Universal Robots PolyScope program: pulley_v2.urp

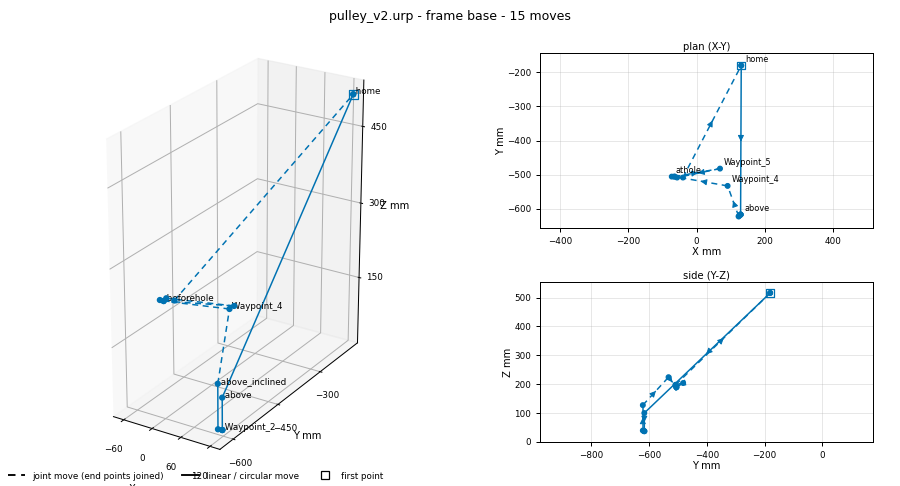
[picture p0: tool path of pulley_v2.urp in frame base, 15 of 23 moves have a stored position in this frame; points joined in program order, loops and branches not executed]
Program pulley_v2 (installation=default directory=/programs/wrs2020 createdIn=5.7.0.90932 lastSavedIn=5.7.0.90932 robotSerialNumber=20205500607)
Calibrated DH parameters: a=[0.000096, -0.337, -0.383372, 0.000118, 0.000015, 0]; d=[0.162724, 79.377998, -95.545185, 16.300583, 0.099689, 0.099499]; alpha=[1.569249, 0.003272, 0.005201, 1.570041, -1.570219, 0]; deltaTheta=[0, 0.65664, 5.410619, 0.215927, -0.000001, 0]
Robot Program (runOnlyOnce=true)
  MoveJ speed 180 deg/s, acceleration 80 deg/s^2 (useActiveTCP=true) feature=Base
    Waypoint home: TCP in base x=130.635 y=-180.692 z=515.97 mm, rx=-0.0117 ry=-3.1402 rz=-0.0315 rad; joints [89.951, -120.324, 80.212, -48.705, -89.957, -0.002] deg; TCP offset x=0 y=0 z=165 mm, rx=0 ry=0 rz=0 rad
  URCap Gripper (Robotiq_Grippers, Robotiq Inc.) dataModel(position=15.686274509803921, force=100.0, speed=100.0, positionInDouble=15.686274509803921, forceInDouble=100.0, speedInDouble=100.0, slaveIds=[9], blocking=true)
  MoveL speed 250 mm/s, acceleration 1200 mm/s^2 (useActiveTCP=true) feature=Base
    Waypoint above: TCP in base x=128.76 y=-616.729 z=99.924 mm, rx=1.2479 ry=2.8551 rz=-0.0099 rad; joints [89.154, -66.805, 95.766, -119.835, -88.426, 46.424] deg
    Waypoint Waypoint_2: TCP in base x=128.767 y=-616.702 z=37 mm, rx=1.2363 ry=2.8602 rz=-0.01 rad; joints [89.14, -62.119, 99.446, -128.198, -88.435, 45.999] deg; TCP offset x=0 y=0 z=165 mm, rx=0 ry=0 rz=0 rad
  URCap Gripper (Robotiq_Grippers, Robotiq Inc.) dataModel(position=100.0, force=0.0, speed=0.0, positionInDouble=100.0, forceInDouble=0.0, speedInDouble=0.0, slaveIds=[9], blocking=true)
  URCap Gripper (Robotiq_Grippers, Robotiq Inc.) dataModel(position=21.176470588235293, force=0.0, speed=0.0, positionInDouble=21.176470588235293, forceInDouble=0.0, speedInDouble=0.0, slaveIds=[9], blocking=true)
  MoveL speed 600 mm/s, acceleration 1200 mm/s^2 (useActiveTCP=true) feature=Base
    Waypoint Waypoint_3: TCP in base x=128.76 y=-616.729 z=37 mm, rx=-1.1525 ry=2.9078 rz=-0.0355 rad; joints [89.139, -62.118, 99.445, -128.202, -88.435, -43.999] deg; TCP offset x=0 y=0 z=165 mm, rx=0 ry=0 rz=0 rad
  URCap Gripper (Robotiq_Grippers, Robotiq Inc.) dataModel(position=100.0, force=0.0, speed=0.0, positionInDouble=100.0, forceInDouble=0.0, speedInDouble=0.0, slaveIds=[9], blocking=true)
  URCap Gripper (Robotiq_Grippers, Robotiq Inc.) dataModel(position=36.07843137254902, force=0.0, speed=0.0, positionInDouble=36.07843137254902, forceInDouble=0.0, speedInDouble=0.0, slaveIds=[9], blocking=true)
  MoveL speed 600 mm/s, acceleration 1200 mm/s^2 (useActiveTCP=true) feature=Base
    Waypoint Waypoint_2: TCP in base x=128.767 y=-616.702 z=37 mm, rx=1.2363 ry=2.8602 rz=-0.01 rad; joints [89.14, -62.119, 99.446, -128.198, -88.435, 45.999] deg; TCP offset x=0 y=0 z=165 mm, rx=0 ry=0 rz=0 rad
    Waypoint Waypoint_1: TCP in base x=123.202 y=-621.873 z=39.247 mm, rx=-1.1443 ry=-2.5469 rz=0.8367 rad; joints [100.881, -59.401, 111.69, -163.652, -118.977, 53.915] deg; TCP offset x=0 y=0 z=165 mm, rx=0 ry=0 rz=0 rad
  URCap Gripper (Robotiq_Grippers, Robotiq Inc.) dataModel(position=100.0, force=100.0, speed=100.0, positionInDouble=100.0, forceInDouble=100.0, speedInDouble=100.0, slaveIds=[9], blocking=true)
  MoveL speed 250 mm/s, acceleration 1200 mm/s^2 (useActiveTCP=true) feature=Base
    Waypoint above_inclined: TCP in base x=123.202 y=-621.873 z=127.29 mm, rx=-1.1443 ry=-2.5469 rz=0.8367 rad; joints [100.905, -68.525, 108.499, -151.362, -118.935, 53.865] deg
  SuppressedNode
    MoveJ speed 60 deg/s, acceleration 80 deg/s^2 (useActiveTCP=true) feature=Base
      Waypoint intermediate: motionParameters(blendRadius=0.05); TCP in base x=115.537 y=-464.392 z=278.491 mm, rx=2.1151 ry=-1.8246 rz=-0.1767 rad; joints [98.791, -95.537, 106.25, -108.287, -109.219, -91.027] deg
      Waypoint before_hole: TCP in base x=-57.686 y=-570.408 z=232.23 mm, rx=1.3727 ry=-1.1616 rz=-1.3181 rad; joints [97.319, -59.573, 88.654, -50.464, -171.504, -31.295] deg
  SuppressedNode
    MoveJ speed 60 deg/s, acceleration 80 deg/s^2 (useActiveTCP=true) feature=Base
      Waypoint at_hole: TCP in base x=-85.495 y=-570.408 z=232.23 mm, rx=1.3727 ry=-1.1616 rz=-1.3181 rad; joints [94.632, -61.815, 93.453, -62.169, -173.913, -40.501] deg; TCP offset x=0 y=0 z=165 mm, rx=0 ry=0 rz=0 rad
  SuppressedNode
    Force Frame feature=Joint_6_name; selection=[0, 0, 1, 0, 0, 0]; wrench=[0, 0, 10, 0, 0, 0]; limitsForce=[0.15, 0.15, 0.01, 1.047198, 1.047198, 1.047198]; limitsMotion=[0.1, 0.1, 0.1, 0.349066, 0.349066, 0.349066]
      MoveJ speed 60 deg/s, acceleration 80 deg/s^2 (useActiveTCP=true) feature=Base
        Waypoint turn_right (Relative): relativeFromPosition TCP in base x=-85.515 y=-570.41 z=232.207 mm, rx=1.3727 ry=-1.1616 rz=-1.3181 rad; joints [94.63, -61.813, 93.454, -62.171, -173.913, -40.501] deg; TCP offset x=0 y=0 z=165 mm, rx=0 ry=0 rz=0 rad; TCP in base x=-85.507 y=-570.407 z=232.241 mm, rx=0.846 ry=-1.441 rz=-0.7763 rad; joints [94.699, -63.491, 97.916, -73.842, -175.626, -8.792] deg
        Waypoint turn_left (Relative): relativeFromPosition TCP in base x=-85.52 y=-570.402 z=232.224 mm, rx=0.846 ry=-1.4411 rz=-0.7763 rad; joints [94.698, -63.49, 97.916, -73.843, -175.624, -8.792] deg; TCP in base x=-85.509 y=-570.398 z=232.173 mm, rx=1.3728 ry=-1.1615 rz=-1.3182 rad; joints [94.631, -61.811, 93.456, -62.169, -173.913, -40.501] deg
        Waypoint turn_left (Relative): relativeFromPosition TCP in base x=-85.52 y=-570.402 z=232.224 mm, rx=0.846 ry=-1.4411 rz=-0.7763 rad; joints [94.698, -63.49, 97.916, -73.843, -175.624, -8.792] deg; TCP in base x=-85.509 y=-570.398 z=232.173 mm, rx=1.3728 ry=-1.1615 rz=-1.3182 rad; joints [94.631, -61.811, 93.456, -62.169, -173.913, -40.501] deg
        Waypoint turn_right (Relative): relativeFromPosition TCP in base x=-85.515 y=-570.41 z=232.207 mm, rx=1.3727 ry=-1.1616 rz=-1.3181 rad; joints [94.63, -61.813, 93.454, -62.171, -173.913, -40.501] deg; TCP in base x=-85.507 y=-570.407 z=232.241 mm, rx=0.846 ry=-1.441 rz=-0.7763 rad; joints [94.699, -63.491, 97.916, -73.842, -175.626, -8.792] deg
  MoveJ speed 120 deg/s, acceleration 150 deg/s^2 (useActiveTCP=true) feature=Base
    Waypoint Waypoint_4: motionParameters(blendRadius=0.05); TCP in base x=90.784 y=-532.798 z=224.095 mm, rx=1.3194 ry=-2.4664 rz=0.0869 rad; joints [93.539, -87.4, 107.422, -121.697, -105.954, -54.416] deg
    Waypoint beforehole: TCP in base x=-64.521 y=-505.594 z=189.248 mm, rx=1.6358 ry=-1.672 rz=-0.8845 rad; joints [92.147, -76.667, 111.26, -118.048, -144.223, -83.204] deg
  MoveL speed 20 mm/s, acceleration 1200 mm/s^2 (useActiveTCP=true) feature=Base
    Waypoint athole: TCP in base x=-72.578 y=-505.587 z=189.228 mm, rx=1.6358 ry=-1.672 rz=-0.8845 rad; joints [91.256, -76.788, 111.802, -119.703, -144.314, -84.72] deg
  MoveL speed 250 mm/s, acceleration 1200 mm/s^2 (useActiveTCP=true) feature=Base
    MoveDirectionNode (selectedDirection=XMinus) feature=Base
      Until TOOL_CONTACT_DETECTION (allowActions=false retraction=0 decelerationAcceleration=3 decelerationAngularAcceleration=34.906585)
  Force Frame feature=Base; selection=[1, 1, 1, 0, 0, 0]; wrench=[-10, 0, 0, 0, 0, 0]; limitsForce=[0.01, 0.01, 0.01, 1.047198, 1.047198, 1.047198]; limitsMotion=[0.1, 0.1, 0.1, 0.349066, 0.349066, 0.349066]
    MoveL speed 50 mm/s, acceleration 200 mm/s^2 (useActiveTCP=true) feature=Base
      Waypoint rightturn (Relative): relativeFromPosition TCP in base x=-72.572 y=-505.592 z=189.212 mm, rx=1.6359 ry=-1.672 rz=-0.8845 rad; joints [91.257, -76.786, 111.802, -119.705, -144.314, -84.72] deg; TCP in base x=-72.593 y=-509.312 z=189.314 mm, rx=1.2962 ry=-1.7188 rz=-0.4228 rad; joints [91.397, -77.772, 124.92, -159.613, -145.042, -84.31] deg
      Waypoint leftturn (Relative): relativeFromPosition TCP in base x=-72.61 y=-509.315 z=189.348 mm, rx=1.2962 ry=-1.7188 rz=-0.4228 rad; joints [91.396, -77.774, 124.918, -159.612, -145.044, -84.311] deg; TCP in base x=-72.577 y=-505.577 z=189.198 mm, rx=1.6359 ry=-1.6719 rz=-0.8846 rad; joints [91.257, -76.786, 111.804, -119.704, -144.316, -84.721] deg
      Waypoint leftturn (Relative): relativeFromPosition TCP in base x=-72.61 y=-509.315 z=189.348 mm, rx=1.2962 ry=-1.7188 rz=-0.4228 rad; joints [91.396, -77.774, 124.918, -159.612, -145.044, -84.311] deg; TCP in base x=-72.577 y=-505.577 z=189.198 mm, rx=1.6359 ry=-1.6719 rz=-0.8846 rad; joints [91.257, -76.786, 111.804, -119.704, -144.316, -84.721] deg
      Waypoint rightturn (Relative): relativeFromPosition TCP in base x=-72.572 y=-505.592 z=189.212 mm, rx=1.6359 ry=-1.672 rz=-0.8845 rad; joints [91.257, -76.786, 111.802, -119.705, -144.314, -84.72] deg; TCP in base x=-72.593 y=-509.312 z=189.314 mm, rx=1.2962 ry=-1.7188 rz=-0.4228 rad; joints [91.397, -77.772, 124.92, -159.613, -145.042, -84.31] deg
  URCap Gripper (Robotiq_Grippers, Robotiq Inc.) dataModel(position=0.0, force=100.0, speed=100.0, positionInDouble=0.0, forceInDouble=100.0, speedInDouble=100.0, slaveIds=[9], blocking=true)
  MoveJ speed 120 deg/s, acceleration 150 deg/s^2 (useActiveTCP=true) feature=Base
    Waypoint beforehole: TCP in base x=-64.521 y=-505.594 z=189.248 mm, rx=1.6358 ry=-1.672 rz=-0.8845 rad; joints [92.147, -76.667, 111.26, -118.048, -144.223, -83.204] deg
    Waypoint Waypoint_5: motionParameters(blendRadius=0.05); TCP in base x=68.522 y=-482.203 z=203.802 mm, rx=1.8496 ry=-2.2565 rz=0.2806 rad; joints [82.53, -98.422, 121.376, -129.22, -89.967, -86.171] deg
    Waypoint Waypoint_8: TCP in base x=-56.985 y=-508.361 z=197.658 mm, rx=1.9455 ry=-2.0776 rz=0.1274 rad; joints [70.293, -94.264, 119.255, -132.207, -92.763, -106.364] deg
  URCap Gripper (Robotiq_Grippers, Robotiq Inc.) dataModel(position=70.58823529411765, force=0.0, speed=0.0, positionInDouble=70.58823529411765, forceInDouble=0.0, speedInDouble=0.0, slaveIds=[9], blocking=true)
  Folder Folder
    loop_1 := 1
    tcp_p := get_actual_tcp_pose()
    Force Frame feature=Base; selection=[1, 0, 0, 0, 0, 0]; wrench=[-10, 0, 0, 0, 0, 0]; limitsForce=[0.01, 0.01, 0.01, 1.047198, 1.047198, 1.047198]; limitsMotion=[0.1, 0.1, 0.1, 0.349066, 0.349066, 0.349066]
      Loop While (checkContinuously=true) expression=( tcp_p[0] > -0.090) and  (loop_1 < 3)
        MoveL speed 50 mm/s, acceleration 200 mm/s^2 (useActiveTCP=true) feature=Base
          Waypoint right1 (Relative): relativeFromPosition TCP in base x=-56.979 y=-508.359 z=197.636 mm, rx=1.9455 ry=-2.0777 rz=0.1274 rad; joints [70.294, -94.262, 119.256, -132.208, -92.762, -106.364] deg; TCP in base x=-56.977 y=-508.344 z=197.639 mm, rx=2.0958 ry=-1.919 rz=0.0946 rad; joints [70.293, -94.264, 119.256, -132.205, -92.762, -115.171] deg
          tcp_p := get_actual_tcp_pose()
          Waypoint left1 (Relative): relativeFromPosition TCP in base x=-56.985 y=-508.33 z=197.605 mm, rx=2.0958 ry=-1.919 rz=0.0945 rad; joints [70.293, -94.262, 119.258, -132.206, -92.764, -115.169] deg; TCP in base x=-56.968 y=-508.356 z=197.628 mm, rx=1.9456 ry=-2.0776 rz=0.1273 rad; joints [70.294, -94.261, 119.255, -132.205, -92.762, -106.365] deg
          tcp_p := get_actual_tcp_pose()
          Waypoint left1 (Relative): relativeFromPosition TCP in base x=-56.985 y=-508.33 z=197.605 mm, rx=2.0958 ry=-1.919 rz=0.0945 rad; joints [70.293, -94.262, 119.258, -132.206, -92.764, -115.169] deg; TCP in base x=-56.968 y=-508.356 z=197.628 mm, rx=1.9456 ry=-2.0776 rz=0.1273 rad; joints [70.294, -94.261, 119.255, -132.205, -92.762, -106.365] deg
          tcp_p := get_actual_tcp_pose()
          Waypoint right1 (Relative): relativeFromPosition TCP in base x=-56.979 y=-508.359 z=197.636 mm, rx=1.9455 ry=-2.0777 rz=0.1274 rad; joints [70.294, -94.262, 119.256, -132.208, -92.762, -106.364] deg; TCP in base x=-56.977 y=-508.344 z=197.639 mm, rx=2.0958 ry=-1.919 rz=0.0946 rad; joints [70.293, -94.264, 119.256, -132.205, -92.762, -115.171] deg
          tcp_p := get_actual_tcp_pose()
        loop_1 := loop_1+1
  MoveJ speed 60 deg/s, acceleration 80 deg/s^2 (useActiveTCP=true) feature=Base
    Waypoint back: TCP in base x=-39.842 y=-508.361 z=197.658 mm, rx=1.9455 ry=-2.0776 rz=0.1274 rad; joints [72.514, -94.336, 119.286, -132.039, -93.419, -104.24] deg
  MoveJ speed 180 deg/s, acceleration 80 deg/s^2 (useActiveTCP=true) feature=Base
    Waypoint home: TCP in base x=130.635 y=-180.692 z=515.97 mm, rx=-0.0117 ry=-3.1402 rz=-0.0315 rad; joints [89.951, -120.324, 80.212, -48.705, -89.957, -0.002] deg
